(* PLC project MotorControl_Universal, PLCAutoPilot AI Code Generator 1.5, author PLCAutoPilot AI *)
(* stored: creationDateTime 2026-06-15T17:57:39.733074 *)

PROGRAM MainProgram
  VAR
    START_BTN AT %I0.0 : BOOL;
    STOP_BTN AT %I0.1 : BOOL;
    MOTOR_RUN AT %Q0.0 : BOOL;
    GREEN_LED AT %Q0.1 : BOOL;
  END_VAR

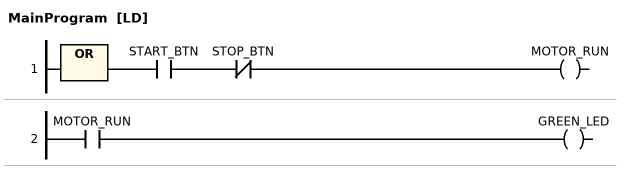
(* LD diagram, written out as Structured Text *)
MOTOR_RUN := OR(TRUE) AND START_BTN AND NOT STOP_BTN;
GREEN_LED := MOTOR_RUN;
END_PROGRAM
